Fanuc KAREL source: ko00021.KL

-- PROVISIONAL review KL for V940-1; original PC SHA256 b54f06943225cfab03b901546d83aab9fa6e39cf848610727b7fdb0f8c89268b
-- Incomplete behavior may be omitted. Consult companion uncertainty JSON. Do not deploy.
PROGRAM KO00021
%NOLOCKGROUP
-- UNRESOLVED_DECL P1 type=000106
-- UNRESOLVED_DECL P2 type=000106
-- UNRESOLVED_DECL P3 type=000106
-- UNRESOLVED_DECL P4 type=000106
-- UNRESOLVED_DECL OUT type=000101
BEGIN
  -- V9_ZERO_TABLE_METADATA_HINT layout=0001; no indexed target words; source/name/runtime held
  -- UNRESOLVED_PC offsets 5-80; opcodes 27,27,49,7E,AD,27,49,7E,AD,27,49,7E,AD,27,49,7E,AD,76,7E,4A
  -- UNRESOLVED_PC offsets 85-89; opcodes 7F
END KO00021
